Yaskawa INFORM job: slope_planes_program.JBI

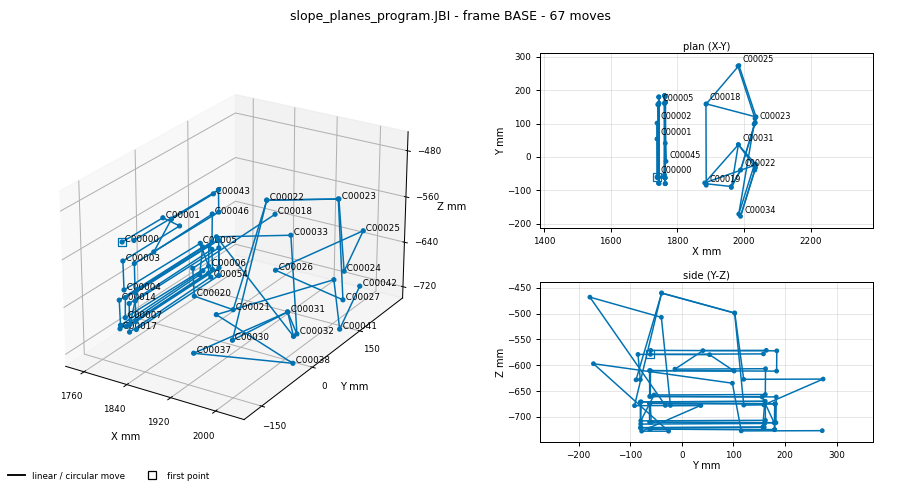
[picture p0: tool path of slope_planes_program.JBI in frame BASE, 67 of 73 moves have a stored position in this frame; points joined in program order, loops and branches not executed]
/JOB
//NAME slope_planes_program
//POS
///NPOS 67,0,67,0,0,0
///TOOL 0
///POSTYPE BASE
///RECTAN
///RCONF 0,0,0,0,0,0,0,0,0,0,0,0,0,0,0,0,0,0,0,0,0,0,0,0
C00000=1739.260769,-60.871235,-578.989580,5.000000,-89.172678,-175.000000
C00001=1739.028106,53.830840,-579.601277,5.000000,-89.172678,-175.000000
C00002=1739.284791,101.372352,-611.275362,5.000000,-89.172678,-175.000000
C00003=1741.092847,-62.556544,-610.379835,5.000000,-89.172678,-175.000000
C00004=1741.778439,-62.282291,-660.377305,5.000000,-89.172678,-175.000000
C00005=1743.760127,155.636241,-661.504448,5.000000,-89.172678,-175.000000
C00006=1744.673230,178.979946,-711.620985,5.000000,-89.172678,-175.000000
C00007=1740.845557,-59.386621,-710.412050,5.000000,-89.172678,-175.000000
C00008=1743.319095,-61.226324,-673.769949,180.000000,-60.000000,0.000000
C00009=1744.726413,180.007491,-675.029042,180.000000,-60.000000,0.000000
C00010=1744.389872,179.342411,-725.036290,180.000000,-60.000000,0.000000
C00011=1744.215946,-60.947521,-723.764393,180.000000,-60.000000,0.000000
C00012=1745.307470,160.600706,-712.870295,175.000000,-89.223717,-5.000000
C00013=1745.747004,-79.714542,-714.068825,175.000000,-89.223717,-5.000000
C00014=1743.887926,-78.841577,-670.993376,180.000000,-60.000000,0.000000
C00015=1744.996879,160.942797,-669.818462,180.000000,-60.000000,0.000000
C00016=1741.316004,156.853693,-719.794086,180.000000,-60.000000,0.000000
C00017=1744.102037,-78.968875,-721.002114,180.000000,-60.000000,0.000000
C00018=1885.863395,158.182403,-578.045584,175.000000,-89.336646,-5.000000
C00019=1886.650424,-84.961125,-579.077831,175.000000,-89.336646,-5.000000
C00020=1886.044276,-80.394228,-627.842130,175.000000,-89.336646,-5.000000
C00021=1961.540570,-88.734620,-628.321589,-5.000000,-89.772434,-156.563433
C00022=1989.769528,-39.136527,-460.340640,175.000000,-47.501225,5.075310
C00023=2033.646978,102.591245,-498.881535,175.000000,-65.273893,-60.828128
C00024=2035.991453,119.891152,-627.326416,175.000000,-89.867726,-65.037930
C00025=1984.737237,273.797954,-626.863225,140.054684,-90.000000,5.000000
C00026=1887.028142,158.913088,-676.850323,175.000000,-89.336646,-5.000000
C00027=2034.825328,120.042378,-677.315653,175.000000,-89.867100,-64.984445
C00028=2032.776243,102.409388,-498.967851,175.000000,-65.312424,-60.640081
C00029=1989.800549,-39.182084,-459.925091,175.000000,-47.287692,5.116560
C00030=1962.013642,-91.664127,-678.436686,5.000000,-89.725460,-155.249492
C00031=1982.938067,36.726704,-677.843770,140.054684,-90.000000,5.000000
C00032=2034.622962,-22.049069,-677.911343,175.000000,-89.867279,-64.999786
C00033=2032.449640,-39.666207,-507.153666,-175.000000,-65.312498,-60.640202
C00034=1989.478498,-178.135948,-468.098074,175.000000,-47.287911,5.116557
C00035=2034.502364,-31.953303,-677.951280,175.000000,-89.866766,-64.955929
C00036=1982.938067,36.726704,-677.843770,140.054684,-90.000000,5.000000
C00037=1882.142247,-77.828377,-727.793743,175.000000,-89.336646,-5.000000
C00038=2030.206063,-25.652685,-727.877558,175.000000,-89.864872,-64.793536
C00039=1984.108354,-171.256741,-597.047291,175.000000,-47.594353,5.056180
C00040=2030.104031,98.022525,-634.851776,-175.000000,-65.256846,-60.910378
C00041=2032.751310,115.122397,-727.316773,-175.000000,-89.868050,-65.065618
C00042=1981.628604,272.117578,-726.841892,140.054684,-90.000000,5.000000
C00043=1764.879905,163.737879,-571.172420,-175.000000,-89.333764,-5.000000
C00044=1764.057547,40.943257,-571.686752,-175.000000,-89.333764,-5.000000
C00045=1766.307154,-13.323645,-607.577811,-175.000000,-89.333764,-5.000000
C00046=1763.380971,162.239603,-606.794756,-175.000000,-89.333764,-5.000000
C00047=1762.810953,161.810268,-656.793795,-175.000000,-89.333764,-5.000000
C00048=1761.795682,-53.749228,-657.701658,-175.000000,-89.333764,-5.000000
C00049=1764.265859,-79.604216,-707.844526,-175.000000,-89.333764,-5.000000
C00050=1763.258444,162.029582,-706.801898,-175.000000,-89.333764,-5.000000
C00051=1762.681818,161.610046,-670.198278,180.000000,-60.000000,0.000000
C00052=1763.869591,-80.392370,-671.244576,180.000000,-60.000000,0.000000
C00053=1763.310066,-80.290661,-721.241471,180.000000,-60.000000,0.000000
C00054=1761.532878,159.749711,-720.196690,180.000000,-60.000000,0.000000
C00055=1761.566018,-60.389450,-571.247562,5.000000,-89.445806,-175.000000
C00056=1761.583926,184.103056,-572.110136,5.000000,-89.445806,-175.000000
C00057=1762.248770,183.727510,-611.406244,5.000000,-89.445806,-175.000000
C00058=1761.627598,-60.731547,-610.549624,5.000000,-89.445806,-175.000000
C00059=1762.073443,-61.075018,-660.546750,5.000000,-89.445806,-175.000000
C00060=1762.413537,182.923131,-661.404463,5.000000,-89.445806,-175.000000
C00061=1763.161347,182.417921,-711.398097,5.000000,-89.445806,-175.000000
C00062=1763.254633,-62.409155,-710.533267,5.000000,-89.445806,-175.000000
C00063=1763.389680,-62.871249,-673.930440,180.000000,-60.000000,0.000000
C00064=1763.610457,181.502527,-674.790632,180.000000,-60.000000,0.000000
C00065=1763.838836,180.206390,-724.786500,180.000000,-60.000000,0.000000
C00066=1763.938440,-62.435048,-723.929321,180.000000,-60.000000,0.000000
///POSTYPE PULSE
///PULSE
EC00000=51200.0
EC00001=51200.0
EC00002=51200.0
EC00003=51200.0
EC00004=51200.0
EC00005=51200.0
EC00006=51200.0
EC00007=51200.0
EC00008=51200.0
EC00009=51200.0
EC00010=51200.0
EC00011=51200.0
EC00012=143360.0
EC00013=143360.0
EC00014=143360.0
EC00015=143360.0
EC00016=143360.0
EC00017=143360.0
EC00018=143360.0
EC00019=143360.0
EC00020=143360.0
EC00021=143360.0
EC00022=143360.0
EC00023=143360.0
EC00024=143360.0
EC00025=143360.0
EC00026=143360.0
EC00027=143360.0
EC00028=143360.0
EC00029=143360.0
EC00030=143360.0
EC00031=143360.0
EC00032=143360.0
EC00033=143360.0
EC00034=143360.0
EC00035=143360.0
EC00036=143360.0
EC00037=143360.0
EC00038=143360.0
EC00039=143360.0
EC00040=143360.0
EC00041=143360.0
EC00042=143360.0
EC00043=235520.0
EC00044=235520.0
EC00045=235520.0
EC00046=235520.0
EC00047=235520.0
EC00048=235520.0
EC00049=235520.0
EC00050=235520.0
EC00051=235520.0
EC00052=235520.0
EC00053=235520.0
EC00054=235520.0
EC00055=327680.0
EC00056=327680.0
EC00057=327680.0
EC00058=327680.0
EC00059=327680.0
EC00060=327680.0
EC00061=327680.0
EC00062=327680.0
EC00063=327680.0
EC00064=327680.0
EC00065=327680.0
EC00066=327680.0
//INST
///DATE 2023/08/13 11:57
///ATTR SC,RW,RJ
////FRAME BASE
///GROUP1 RB1,ST1
NOP
MOVJ P009 EX000 VJ=15.00
MOVJ C00000 EC00000 VJ=15.0
CALL JOB:SPYON
MOVL C00001 EC00001 V=150.0
MOVL C00002 EC00002 V=150.0
MOVL C00003 EC00003 V=150.0
MOVL C00004 EC00004 V=150.0
MOVL C00005 EC00005 V=150.0
MOVL C00006 EC00006 V=150.0
MOVL C00007 EC00007 V=150.0
MOVL C00008 EC00008 V=150.0
MOVL C00009 EC00009 V=150.0
MOVL C00010 EC00010 V=150.0
MOVL C00011 EC00011 V=150.0
CALL JOB:SPYOF
MOVJ P009 VJ=15.00
MOVJ C00012 EC00012 VJ=15.0
CALL JOB:SPYON
MOVL C00013 EC00013 V=150.0
MOVL C00014 EC00014 V=150.0
MOVL C00015 EC00015 V=150.0
MOVL C00016 EC00016 V=150.0
MOVL C00017 EC00017 V=150.0
CALL JOB:SPYOF
MOVJ P009 VJ=15.00
MOVJ C00018 EC00018 VJ=15.0
CALL JOB:SPYON
MOVL C00019 EC00019 V=150.0
MOVL C00020 EC00020 V=150.0
MOVL C00021 EC00021 V=150.0
MOVL C00022 EC00022 V=150.0
MOVL C00023 EC00023 V=150.0
MOVL C00024 EC00024 V=150.0
MOVL C00025 EC00025 V=150.0
MOVL C00026 EC00026 V=150.0
MOVL C00027 EC00027 V=150.0
MOVL C00028 EC00028 V=150.0
MOVL C00029 EC00029 V=150.0
MOVL C00030 EC00030 V=150.0
MOVL C00031 EC00031 V=150.0
MOVL C00032 EC00032 V=150.0
MOVL C00033 EC00033 V=150.0
MOVL C00034 EC00034 V=150.0
MOVL C00035 EC00035 V=150.0
MOVL C00036 EC00036 V=150.0
MOVL C00037 EC00037 V=150.0
MOVL C00038 EC00038 V=150.0
MOVL C00039 EC00039 V=150.0
MOVL C00040 EC00040 V=150.0
MOVL C00041 EC00041 V=150.0
MOVL C00042 EC00042 V=150.0
CALL JOB:SPYOF
MOVJ P009 VJ=15.00
MOVJ C00043 EC00043 VJ=15.0
CALL JOB:SPYON
MOVL C00044 EC00044 V=150.0
MOVL C00045 EC00045 V=150.0
MOVL C00046 EC00046 V=150.0
MOVL C00047 EC00047 V=150.0
MOVL C00048 EC00048 V=150.0
MOVL C00049 EC00049 V=150.0
MOVL C00050 EC00050 V=150.0
MOVL C00051 EC00051 V=150.0
MOVL C00052 EC00052 V=150.0
MOVL C00053 EC00053 V=150.0
MOVL C00054 EC00054 V=150.0
CALL JOB:SPYOF
MOVJ P009 VJ=15.00
MOVJ C00055 EC00055 VJ=15.0
CALL JOB:SPYON
MOVL C00056 EC00056 V=150.0
MOVL C00057 EC00057 V=150.0
MOVL C00058 EC00058 V=150.0
MOVL C00059 EC00059 V=150.0
MOVL C00060 EC00060 V=150.0
MOVL C00061 EC00061 V=150.0
MOVL C00062 EC00062 V=150.0
MOVL C00063 EC00063 V=150.0
MOVL C00064 EC00064 V=150.0
MOVL C00065 EC00065 V=150.0
MOVL C00066 EC00066 V=150.0
CALL JOB:SPYOF
MOVJ P009 VJ=15.00
END
